FUNCTION_BLOCK DeliveryServices_Adp (* Composite Function Block Type *)
  (* Standard: 61499-2 *)
  (* Version 0.0, 11/25/2020, prana, nxtControl GmbH, template *)
  PACKAGE Main;
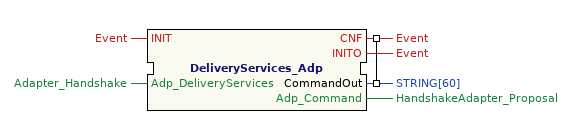
  EVENT_INPUT
    INIT; (* Initialization Request *)
  END_EVENT
  EVENT_OUTPUT
    CNF WITH CommandOut; (* Execution Confirmation *)
    INITO; (* Initialization Confirm *)
  END_EVENT
  VAR_OUTPUT
    CommandOut : STRING[60]; (* Output event qualifier *)
  END_VAR
  SOCKETS
    Adp_DeliveryServices : Adapter_Handshake;
  END_SOCKETS
  PLUGS
    Adp_Command : HandshakeAdapter_Proposal;
  END_PLUGS
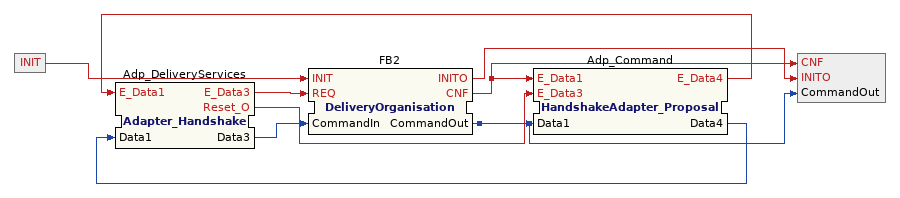
  FBS
    FB2 : DeliveryOrganisation;
  END_FBS
  EVENT_CONNECTIONS
    Adp_Command.E_Data4 TO Adp_DeliveryServices.E_Data1;
    FB2.CNF TO Adp_Command.E_Data1;
    FB2.CNF TO CNF;
    Adp_DeliveryServices.E_Data3 TO FB2.REQ;
    INIT TO FB2.INIT;
    FB2.INITO TO INITO;
    Adp_DeliveryServices.Reset_O TO Adp_Command.E_Data3;
  END_CONNECTIONS
  DATA_CONNECTIONS
    Adp_Command.Data4 TO Adp_DeliveryServices.Data1;
    FB2.CommandOut TO Adp_Command.Data1;
    FB2.CommandOut TO CommandOut;
    Adp_DeliveryServices.Data3 TO FB2.CommandIn;
  END_CONNECTIONS
END_FUNCTION_BLOCK
